(* IEC 61131-3 sources: matiec/tests/string_widths, 24 files *)

(* ---- bounded_il_reject.st ---- *)
FUNCTION_BLOCK FB1
  VAR
    X : STRING[10];
  END_VAR
  LD X
  ST X
END_FUNCTION_BLOCK

PROGRAM prog0
  VAR
    F : FB1;
  END_VAR
  F();
END_PROGRAM

CONFIGURATION config
  RESOURCE res ON PLC
    TASK tsk(INTERVAL := T#100ms, PRIORITY := 0);
    PROGRAM inst0 WITH tsk : prog0;
  END_RESOURCE
END_CONFIGURATION

(* ---- bounded_inout.st ---- *)
FUNCTION_BLOCK FB1
  VAR_IN_OUT
    S : STRING;
  END_VAR
  S := 'abcdefghijklmno';
END_FUNCTION_BLOCK

PROGRAM prog0
  VAR
    F : FB1;
    N : STRING[10];
  END_VAR
  F(S := N);
END_PROGRAM

CONFIGURATION config
  RESOURCE res ON PLC
    TASK tsk(INTERVAL := T#100ms, PRIORITY := 0);
    PROGRAM inst0 WITH tsk : prog0;
  END_RESOURCE
END_CONFIGURATION

(* ---- bounded_out_param.st ---- *)
FUNCTION_BLOCK FB1
  VAR_OUTPUT
    O : STRING;
  END_VAR
  O := 'abcdefghijklmno';
END_FUNCTION_BLOCK

PROGRAM prog0
  VAR
    F : FB1;
    N : STRING[10];
  END_VAR
  F(O => N);
END_PROGRAM

CONFIGURATION config
  RESOURCE res ON PLC
    TASK tsk(INTERVAL := T#100ms, PRIORITY := 0);
    PROGRAM inst0 WITH tsk : prog0;
  END_RESOURCE
END_CONFIGURATION

(* ---- fb_bounded.st ---- *)
FUNCTION_BLOCK FB1
  VAR_INPUT
    NAME : STRING[15];
  END_VAR
  VAR_OUTPUT
    OUT : STRING;
  END_VAR
  OUT := NAME;
END_FUNCTION_BLOCK

PROGRAM prog0
  VAR
    F : FB1;
    S : STRING := 'abcdefghijklmnopqrstuvwxyz';
    R : STRING;
    M : STRING;
  END_VAR
  F(NAME := S);
  R := F.OUT;
  M := F.NAME;
END_PROGRAM

CONFIGURATION config
  RESOURCE res ON PLC
    TASK tsk(INTERVAL := T#100ms, PRIORITY := 0);
    PROGRAM inst0 WITH tsk : prog0;
  END_RESOURCE
END_CONFIGURATION

(* ---- struct_bounded_out_param.st ---- *)
(* C4 parity: a bounded struct member receiving a function block output behaves
 * exactly as the bounded variable in bounded_out_param does - a truncating
 * __SET_STRVAR at the declared width, not an unchecked copy.
 *)
TYPE
  REC : STRUCT
    F : STRING[10];
  END_STRUCT;
END_TYPE

FUNCTION_BLOCK SRC
VAR_OUTPUT
  O : STRING;
END_VAR
  O := 'abcdefghijklmno';
END_FUNCTION_BLOCK

PROGRAM prog0
  VAR
    R : REC;
    S : SRC;
  END_VAR
  S(O => R.F);
END_PROGRAM

CONFIGURATION config
  RESOURCE res ON PLC
    TASK tsk(INTERVAL := T#100ms, PRIORITY := 0);
    PROGRAM inst0 WITH tsk : prog0;
  END_RESOURCE
END_CONFIGURATION

(* ---- struct_nested_access.st ---- *)
(* R4: narrowing writes and widening reads through a direct member, a member of a
 * nested struct, and a struct passed as a FUNCTION_BLOCK input - the DISPLAY4 shape.
 *)
TYPE
  INNER : STRUCT
    D : STRING[10];
  END_STRUCT;
  OUTER : STRUCT
    I : INNER;
    T : STRING[10];
  END_STRUCT;
END_TYPE

FUNCTION_BLOCK SINK
VAR_INPUT
  LINE : INNER;
END_VAR
VAR_OUTPUT
  SEEN : STRING;
END_VAR
  SEEN := LINE.D;
END_FUNCTION_BLOCK

PROGRAM prog0
  VAR
    WIDE : STRING := '123456789012345678901234567890';
    O    : OUTER;
    S    : SINK;
    BACK : STRING;
  END_VAR
  O.T   := WIDE;
  O.I.D := WIDE;
  BACK  := O.I.D;
  S(LINE := O.I);
END_PROGRAM

CONFIGURATION config
  RESOURCE res ON PLC
    TASK tsk(INTERVAL := T#100ms, PRIORITY := 0);
    PROGRAM inst0 WITH tsk : prog0;
  END_RESOURCE
END_CONFIGURATION

(* ---- assign_narrow.st ---- *)
PROGRAM prog0
  VAR
    WIDE   : STRING := '123456789012345678901234567890';
    NARROW : STRING[10];
    OUT    : STRING;
  END_VAR
  NARROW := WIDE;
  OUT := NARROW;
  OUT := CONCAT(NARROW, 'X');
END_PROGRAM

CONFIGURATION config
  RESOURCE res ON PLC
    TASK tsk(INTERVAL := T#100ms, PRIORITY := 0);
    PROGRAM inst0 WITH tsk : prog0;
  END_RESOURCE
END_CONFIGURATION

(* ---- bounded_decl.st ---- *)
PROGRAM prog0
  VAR
    A : STRING[20];
    B : STRING[20] := 'hi';
  END_VAR
  A := B;
END_PROGRAM

CONFIGURATION config
  RESOURCE res ON PLC
    TASK tsk(INTERVAL := T#100ms, PRIORITY := 0);
    PROGRAM inst0 WITH tsk : prog0;
  END_RESOURCE
END_CONFIGURATION

(* ---- bounded_fn_local_out.st ---- *)
FUNCTION FN2 : INT
  VAR_INPUT
    I : INT;
  END_VAR
  VAR_OUTPUT
    O : STRING;
  END_VAR
  O := 'abcdefghijklmno';
  FN2 := I;
END_FUNCTION

FUNCTION FN1 : INT
  VAR_INPUT
    J : INT;
  END_VAR
  VAR
    X : STRING[10];
    R : INT;
  END_VAR
  R := FN2(I := J, O => X);
  FN1 := R;
END_FUNCTION

PROGRAM prog0
  VAR
    R : INT;
  END_VAR
  R := FN1(1);
END_PROGRAM

CONFIGURATION config
  RESOURCE res ON PLC
    TASK tsk(INTERVAL := T#100ms, PRIORITY := 0);
    PROGRAM inst0 WITH tsk : prog0;
  END_RESOURCE
END_CONFIGURATION

(* ---- bounded_fn_out.st ---- *)
FUNCTION FN1 : INT
  VAR_INPUT
    I : INT;
  END_VAR
  VAR_OUTPUT
    O : STRING;
  END_VAR
  O := 'abcdefghijklmno';
  FN1 := I;
END_FUNCTION

PROGRAM prog0
  VAR
    N : STRING[10];
    R : INT;
  END_VAR
  R := FN1(I := 1, O => N);
END_PROGRAM

CONFIGURATION config
  RESOURCE res ON PLC
    TASK tsk(INTERVAL := T#100ms, PRIORITY := 0);
    PROGRAM inst0 WITH tsk : prog0;
  END_RESOURCE
END_CONFIGURATION

(* ---- escaped_literal.st ---- *)
PROGRAM prog0
  VAR
    A : STRING[3] := 'a$Tb';
    B : STRING[2] := '$$$'';
  END_VAR
  A := A;
END_PROGRAM

CONFIGURATION config
  RESOURCE res ON PLC
    TASK tsk(INTERVAL := T#100ms, PRIORITY := 0);
    PROGRAM inst0 WITH tsk : prog0;
  END_RESOURCE
END_CONFIGURATION

(* ---- fn_bounded_body.st ---- *)
(* Bounded strings inside a FUNCTION body: its variables are plain C objects, so the
 * accessor macros that normally carry the widen/narrow conversions do not apply.
 * Covers a bounded local and a bounded member of the function's return value.
 *)
TYPE
  REC : STRUCT
    F : STRING[10];
  END_STRUCT;
END_TYPE

FUNCTION MAKE_REC : REC
VAR_INPUT
  S : STRING;
END_VAR
VAR
  B : STRING[10];
END_VAR
  B := S;
  MAKE_REC.F := B;
END_FUNCTION

PROGRAM prog0
VAR
  R : REC;
END_VAR
  R := MAKE_REC(S := '123456789012345');
END_PROGRAM

CONFIGURATION config
  RESOURCE res ON PLC
    TASK tsk(INTERVAL := T#100ms, PRIORITY := 0);
    PROGRAM inst0 WITH tsk : prog0;
  END_RESOURCE
END_CONFIGURATION

(* ---- global_bounded.st ---- *)
PROGRAM prog0
  VAR_EXTERNAL
    G : STRING;
  END_VAR
  G := 'x';
END_PROGRAM

CONFIGURATION config
  VAR_GLOBAL
    G : STRING[12];
  END_VAR
  RESOURCE res ON PLC
    TASK tsk(INTERVAL := T#100ms, PRIORITY := 0);
    PROGRAM inst0 WITH tsk : prog0;
  END_RESOURCE
END_CONFIGURATION

(* ---- overlong_literal.st ---- *)
PROGRAM prog0
  VAR
    A : STRING[20] := '123456789012345678901234567890';
  END_VAR
  A := A;
END_PROGRAM

CONFIGURATION config
  RESOURCE res ON PLC
    TASK tsk(INTERVAL := T#100ms, PRIORITY := 0);
    PROGRAM inst0 WITH tsk : prog0;
  END_RESOURCE
END_CONFIGURATION

(* ---- plain_string.st ---- *)
PROGRAM prog0
  VAR
    A : STRING;
    B : STRING := 'hello';
  END_VAR
  A := B;
END_PROGRAM

CONFIGURATION config
  RESOURCE res ON PLC
    TASK tsk(INTERVAL := T#100ms, PRIORITY := 0);
    PROGRAM inst0 WITH tsk : prog0;
  END_RESOURCE
END_CONFIGURATION

(* ---- struct_bounded_init.st ---- *)
(* Bounded counterpart of struct_plain_init: member default, no default, and a
 * per-instance initializer, all at a declared width. Any difference in behaviour
 * between the two fixtures is attributable to STRING[n].
 *)
TYPE
  REC : STRUCT
    F : STRING[10] := 'abc';
    G : STRING[10];
    N : INT := 7;
  END_STRUCT;
END_TYPE

PROGRAM prog0
  VAR
    R1 : REC;
    R2 : REC := (F := 'xy', N := 9);
  END_VAR
  R1.N := R1.N;
END_PROGRAM

CONFIGURATION config
  RESOURCE res ON PLC
    TASK tsk(INTERVAL := T#100ms, PRIORITY := 0);
    PROGRAM inst0 WITH tsk : prog0;
  END_RESOURCE
END_CONFIGURATION

(* ---- struct_bounded_var.st ---- *)
(* A variable of a struct type with a bounded member: storage is the declared
 * width and the member default-initialises empty.
 *)
TYPE
  REC : STRUCT
    F : STRING[10];
    N : INT;
  END_STRUCT;
END_TYPE

PROGRAM prog0
  VAR
    R : REC;
  END_VAR
  R.N := 1;
END_PROGRAM

CONFIGURATION config
  RESOURCE res ON PLC
    TASK tsk(INTERVAL := T#100ms, PRIORITY := 0);
    PROGRAM inst0 WITH tsk : prog0;
  END_RESOURCE
END_CONFIGURATION

(* ---- struct_overlong_default.st ---- *)
(* R6: a member default longer than the declared width is a build error,
 * not a silent truncation.
 *)
TYPE
  REC : STRUCT
    F : STRING[10] := 'ABCDEFGHIJK';
  END_STRUCT;
END_TYPE

PROGRAM prog0
  VAR
    R : REC;
  END_VAR
  R.F := R.F;
END_PROGRAM

CONFIGURATION config
  RESOURCE res ON PLC
    TASK tsk(INTERVAL := T#100ms, PRIORITY := 0);
    PROGRAM inst0 WITH tsk : prog0;
  END_RESOURCE
END_CONFIGURATION

(* ---- struct_plain_init.st ---- *)
(* Pre-existing behaviour probe: a plain (unbounded) STRING as a TYPE...STRUCT member,
 * with a member default, without one, and overridden by a per-instance initializer.
 * No STRING[n] anywhere - this must already work before X-37a builds on it.
 *)
TYPE
  REC : STRUCT
    F : STRING := 'abc';
    G : STRING;
    N : INT := 7;
  END_STRUCT;
END_TYPE

PROGRAM prog0
  VAR
    R1 : REC;
    R2 : REC := (F := 'xy', N := 9);
  END_VAR
  R1.N := R1.N;
END_PROGRAM

CONFIGURATION config
  RESOURCE res ON PLC
    TASK tsk(INTERVAL := T#100ms, PRIORITY := 0);
    PROGRAM inst0 WITH tsk : prog0;
  END_RESOURCE
END_CONFIGURATION

(* ---- width_max.st ---- *)
PROGRAM prog0
  VAR
    A : STRING[126];
  END_VAR
  A := A;
END_PROGRAM

CONFIGURATION config
  RESOURCE res ON PLC
    TASK tsk(INTERVAL := T#100ms, PRIORITY := 0);
    PROGRAM inst0 WITH tsk : prog0;
  END_RESOURCE
END_CONFIGURATION

(* ---- width_too_large.st ---- *)
PROGRAM prog0
  VAR
    A : STRING[127];
  END_VAR
  A := A;
END_PROGRAM

CONFIGURATION config
  RESOURCE res ON PLC
    TASK tsk(INTERVAL := T#100ms, PRIORITY := 0);
    PROGRAM inst0 WITH tsk : prog0;
  END_RESOURCE
END_CONFIGURATION

(* ---- width_underscore.st ---- *)
PROGRAM prog0
  VAR
    A : STRING[1_00];
  END_VAR
  A := A;
END_PROGRAM

CONFIGURATION config
  RESOURCE res ON PLC
    TASK tsk(INTERVAL := T#100ms, PRIORITY := 0);
    PROGRAM inst0 WITH tsk : prog0;
  END_RESOURCE
END_CONFIGURATION

(* ---- width_underscore_rejected.st ---- *)
PROGRAM prog0
  VAR
    A : STRING[1_27];
  END_VAR
  A := A;
END_PROGRAM

CONFIGURATION config
  RESOURCE res ON PLC
    TASK tsk(INTERVAL := T#100ms, PRIORITY := 0);
    PROGRAM inst0 WITH tsk : prog0;
  END_RESOURCE
END_CONFIGURATION

(* ---- width_zero.st ---- *)
PROGRAM prog0
  VAR
    A : STRING[0];
  END_VAR
  A := A;
END_PROGRAM

CONFIGURATION config
  RESOURCE res ON PLC
    TASK tsk(INTERVAL := T#100ms, PRIORITY := 0);
    PROGRAM inst0 WITH tsk : prog0;
  END_RESOURCE
END_CONFIGURATION
